FUNCTION alg_M_example_controller_a_Dstartled : BOOL
VAR_INPUT
	state: STATE;
END_VAR

alg_M_example_controller_a_Dstartled := (state.dvar_M_example_controller) = (elit_wait_start);

END_FUNCTION

(* stored: Version 1.1.0.1, ProductVersion 3.1.4022.18
   POU alg_M_example_controller_a_Dstartled: Id {783a29b5-c33c-4ac8-ae29-45d8d8a9c3f0}, SpecialFunc None *)
